PROGRAM MAIN
VAR
	fbCar : FB_Car := (fFuelKilometerLimit := 4853453645);
	fbEngine : FB_PetrolEngine;
	bStart : BOOL;
	bDrive : BOOL;
END_VAR


IF bStart THEN
	fbCar.Start();
	fbCar(fbEngine := fbEngine);
END_IF

END_PROGRAM

(* stored: Version 1.1.0.1, ProductVersion 3.1.4024.16
   POU MAIN: Id {1eb1897d-6236-408c-b038-5d9babf5f616}, SpecialFunc None *)
